PROGRAM Main
VAR
	// Leica Variables
	AngleHz			AT %I* : LREAL := 0.0;
	AngleVt			AT %I* : LREAL := 0.0;
	Distance		AT %I* : LREAL := 0.0;
	q0				AT %I* : LREAL := 0.0;
	q1				AT %I* : LREAL := 0.0;
	q2				AT %I* : LREAL := 0.0;
	q3				AT %I* : LREAL := 0.0;
	Timestamp		AT %I* : ULINT := 0;
	x				: LREAL := 0.0;
	y				: LREAL := 0.0;
	z				: LREAL := 0.0;
	
	counter			: UDINT := 0;
	
	
	
END_VAR


// Leica transform to x,y and z coordinates
x := Distance*SIN(AngleVt)*SIN(AngleHz);
y := Distance*SIN(AngleVt)*COS(AngleHz);
z := Distance*COS(AngleVt);

counter := counter + 1;

END_PROGRAM

(* stored: Version 1.1.0.1, ProductVersion 3.1.4020.12
   POU Main: Id {841967ed-ee1e-4fd2-acd5-2d10c3ac666f}, SpecialFunc None *)
